KUKA KRL program: ros_rsi_extaxis_v2.src

&ACCESS RVP
&REL 13
&PARAM EDITMASK = *
&PARAM TEMPLATE = C:\KRC\Roboter\Template\vorgabe
DEF ros_rsi( )

; =============================================
;
; Software License Agreement (BSD License)
;
; Copyright (c) 2014 Norwegian University of Science and Technology
; All rights reserved.
;
; Redistribution and use in source and binary forms, with or without
; modification, are permitted provided that the following conditions
; are met:
;
;  * Redistributions of source code must retain the above copyright
;    notice, this list of conditions and the following disclaimer.
;  * Redistributions in binary form must reproduce the above
;    copyright notice, this list of conditions and the following
;    disclaimer in the documentation and/or other materials provided
;    with the distribution.
;  * Neither the name of the Norwegian University of Science and
;    Technology, nor the names of its contributors may be used to
;    endorse or promote products derived from this software without
;    specific prior written permission.
;
; THIS SOFTWARE IS PROVIDED BY THE COPYRIGHT HOLDERS AND CONTRIBUTORS
; "AS IS" AND ANY EXPRESS OR IMPLIED WARRANTIES, INCLUDING, BUT NOT
; LIMITED TO, THE IMPLIED WARRANTIES OF MERCHANTABILITY AND FITNESS
; FOR A PARTICULAR PURPOSE ARE DISCLAIMED. IN NO EVENT SHALL THE
; COPYRIGHT OWNER OR CONTRIBUTORS BE LIABLE FOR ANY DIRECT, INDIRECT,
; INCIDENTAL, SPECIAL, EXEMPLARY, OR CONSEQUENTIAL DAMAGES (INCLUDING,
; BUT NOT LIMITED TO, PROCUREMENT OF SUBSTITUTE GOODS OR SERVICES;
; LOSS OF USE, DATA, OR PROFITS; OR BUSINESS INTERRUPTION) HOWEVER
; CAUSED AND ON ANY THEORY OF LIABILITY, WHETHER IN CONTRACT, STRICT
; LIABILITY, OR TORT (INCLUDING NEGLIGENCE OR OTHERWISE) ARISING IN
; ANY WAY OUT OF THE USE OF THIS SOFTWARE, EVEN IF ADVISED OF THE
; POSSIBILITY OF SUCH DAMAGE.
;
; =============================================

; =============================================
;
; ROS INDUSTRIAL: KUKA RSI HW INTERFACE
; Realtime UDP data exchange with
; kuka_rsi_hw_interface
;
; =============================================

; Declaration of KRL variables
DECL INT ret	; Return value for RSI commands
DECL INT CONTID	; ContainerID

;FOLD INI
  ;FOLD BASISTECH INI
    GLOBAL INTERRUPT DECL 3 WHEN $STOPMESS==TRUE DO IR_STOPM ( )
    INTERRUPT ON 3
    BAS (#INITMOV,0 )
  ;ENDFOLD (BASISTECH INI)
  ;FOLD USER INI
    ;Make your modifications here

  ;ENDFOLD (USER INI)
;ENDFOLD (INI)

; Move to start position


PTP $POS_ACT

; Create RSI Context
ret = RSI_CREATE("ros_rsi_extaxis_v2",CONTID,TRUE)
IF (ret <> RSIOK) THEN
  HALT
ENDIF

; Start RSI execution
ret = RSI_ON(#RELATVIVE)
IF (ret <> RSIOK) THEN
  HALT
ENDIF

;;FOLD WAIT Time= 5.0 sec ;%{PE}
;;FOLD Parameters ;%{h}
;;Params IlfProvider=kukaroboter.basistech.inlineforms.logics.wait; Time=5.0
;;ENDFOLD
;WAIT SEC 5.0
;;ENDFOLD
; Sensor guided movement
RSI_MOVECORR()

; Turn off RSI
ret = RSI_OFF()
IF (ret <> RSIOK) THEN
  HALT
ENDIF


PTP $POS_ACT
END
